Universal Robots PolyScope program: get_information.urp

Program get_information (installation=default directory=/programs createdIn=5.2.0.61336 lastSavedIn=5.2.0.61336 robotSerialNumber=20185300040)
Calibrated DH parameters: a=[-0.000128, -0.221415, -0.194849, 0.000098, -0.000148, 0]; d=[0.152137, 33.879231, 13.968137, -47.716378, 0.085395, 0.092257]; alpha=[1.57105, 0.003021, -0.001826, 1.571145, -1.57192, 0]; deltaTheta=[0, 0.433042, -0.854582, 0.421536, 0.000002, 0]
BeforeStart
  connection := socket_open("10.0.47.214", 30050)
Robot Program (runOnlyOnce=true)
  Loop While (checkContinuously=false) expression=connection≟ False
    connection := socket_open("10.0.47.214", 30050)
    Wait Sleep waitTime=0.5
  Script: socket_send_string("ask_me")
  Wait Sleep waitTime=0.5
  command := socket_read_ascii_float(1)
  Wait Sleep waitTime=0.01
  If command[0] ≠ 0
    Switch expression=command[1]
      Case (caseValue=1)
        response := get_actual_tcp_pose()
      Case (caseValue=2)
        Script: pose = socket_read_string()
        Script: response = is_within_safety_limits(pose)
      Case (caseValue=3)
        Script: register = socket_read_ascii_float(1)
        Script: response = read_port_register(register[1])
      Case (caseValue=4)
        Script: response = is_steady()
      Case (caseValue=2147483647)
        Script: response = "ERROR"
    Script: socket_send_string(response)
  Script: connection = False
  Script: socket_close()
